(* 
:Description: This function block is used represent basic axis controled by standard PLCopen motion function blocks with collision avoidance feature.
*)
FUNCTION_BLOCK FB_AxisServoCA EXTENDS FB_AxisServo IMPLEMENTS I_UniversalAxisCA
VAR
	(*Commands *)
	bHaltCA				: BOOL;	(*  *)
	bMoveAbsoluteCA		: BOOL;	(*  *)
	bMoveRelativeCA		: BOOL;	(*  *)
	bHaltedCA			: BOOL;
	
	(* Parameters *)
	lrGap				: MC_LREAL;
	eDirectionCa		: Tc3_Mc3Definitions.MC_DIRECTION; (* Axis movement direction for collision avoidance *)
	stMoveAbsCaOptions	: ST_MoveAbsoluteCAOptions;
		
	(* Function blocks *)
	fbMcHaltCA			: MC_HaltCA;			(* Halt with colision avoidance *)
	fbMcMoveAbsoluteCA	: MC_MoveAbsoluteCA;	(* Move absolute with colision avoidance *)
	fbMcMoveRelativeCA	: MC_MoveRelativeCA;	(* Move relative with colision avoidance *)
	
	eAxisStateCA		: E_AxisStateCA;		(*  *)
	tonDelay			: TON;				(* Delay which allows to see any page changes during tests *)

END_VAR
(*
Version history:

+-------------+------------+----------------+----------+------------------------------------------+
|Date         | Version    | created under  | Author   | Remark                                   |
+=============+============+================+==========+==========================================+
|2021-11      | 1.0.0.0    | V3.1.4024.22   | ADBO     | Function block created                   |
+-------------+------------+----------------+----------+------------------------------------------+

*)

IF bFirstCycle THEN
	stMoveAbsCaOptions.GapControlMode := MC_GAP_CONTROL_MODE.mcGapControlModeStandard;
END_IF

SUPER^();

tonDelay();

PROPERTY DirectionCA : Tc3_Mc3Definitions.MC_DIRECTION
GET
DirectionCA := eDirectionCa;
END_GET
SET
eDirectionCa := DirectionCA;
END_SET
END_PROPERTY

PROPERTY Gap : MC_LREAL
GET
Gap := lrGap;
END_GET
SET
lrGap := Gap;
END_SET
END_PROPERTY

PROPERTY HaltedCA : REFERENCE TO BOOL
GET
HaltedCA REF= bHaltedCA;
END_GET
END_PROPERTY

METHOD MR_HaltCA : BOOL
VAR_INPUT
END_VAR
IF eAxisState >= AXIS_IDLE AND eAxisStateCA <> AXIS_CA_HALT_DONE THEN
	bHaltedCA := FALSE;
	
	IF NOT bHaltLog THEN 
		fbMachineLogger.MR_AddLogs(CONCAT(sName,' : halt (CA) requested'));
		bHaltLog := TRUE;
	END_IF
	
	bHaltCA := TRUE;
	MR_HaltCA := FALSE;
	eAxisState := AXIS_EXTENSION;
	eAxisStateCA := AXIS_CA_HALT;
	
ELSIF eAxisState = AXIS_EXTENSION AND eAxisStateCA = AXIS_CA_HALT_DONE THEN
	bInPostion 	:= FALSE;
	bInVelocity := FALSE;
	bMoveActive := FALSE;
	bStopped 	:= FALSE;
	bJogDone 	:= FALSE;
	bHaltedCA	:= TRUE;
	
	bHaltCA		:= FALSE;
	MR_HaltCA 	:= TRUE;
	bHaltLog 	:= FALSE;
	fbMachineLogger.MR_AddLogs(CONCAT(sName,' : halt (CA) done'));
	
END_IF
END_METHOD

METHOD MR_MoveAbsoluteCA : BOOL
VAR_INPUT
	lrAbsolutePosition : LREAL;
END_VAR
VAR
	bFirstCycle		   : BOOL := TRUE;
END_VAR
VAR_INST
	lrAbsolutePositionTemp : LREAL;
END_VAR
IF bFirstCycle THEN
	bFirstCycle := FALSE;
	
	IF THIS^.lrAbsolutePosition = lrAbsolutePosition THEN
		lrAbsolutePositionTemp := lrAbsolutePosition - 0.001;
		
	ELSE
		lrAbsolutePositionTemp := lrAbsolutePosition;
		
	END_IF
END_IF


IF eAxisState = AXIS_IDLE AND THIS^.lrAbsolutePosition <> lrAbsolutePositionTemp THEN
	THIS^.lrAbsolutePosition := lrAbsolutePosition;
	bInPostion 	:= FALSE;
	bInVelocity := FALSE;
	bMoveActive := TRUE;
	bStopped 	:= FALSE;
	bHalted 	:= FALSE;
	bJogDone 	:= FALSE;
	bHaltedCA 	:= FALSE;
	
	bMoveAbsoluteCA := TRUE;
	MR_MoveAbsoluteCA := FALSE;
	eAxisState := AXIS_EXTENSION;
	eAxisStateCA := AXIS_CA_MOVE_ABSOLUTE;
	fbMachineLogger.MR_AddLogs(CONCAT(sName,' : move absoulte (CA) requested'));		
	
ELSIF eAxisState = AXIS_EXTENSION AND eAxisStateCA = AXIS_CA_MOVE_ABSOLUTE_DONE THEN
	bInPostion 		:= TRUE;
	bInVelocity		:= FALSE;
	bMoveActive 	:= FALSE;
	bStopped 		:= FALSE;
	bHalted			:= FALSE;
	bJogDone 		:= FALSE;
	bHaltedCA 		:= TRUE;
	
	bMoveAbsoluteCA := FALSE;
	MR_MoveAbsoluteCA := TRUE;
	fbMachineLogger.MR_AddLogs(CONCAT(sName,' : move absoulte (CA) done'));		
	
END_IF
END_METHOD

METHOD MR_MoveRelativeCA : BOOL
VAR_INPUT
	lrRelativeDistance : LREAL;
END_VAR
IF eAxisState = AXIS_IDLE AND lrRelativeDistance <> 0.0 THEN
	bInPostion 	:= FALSE;
	
	THIS^.lrRelativeDistance := lrRelativeDistance;
	bInVelocity := FALSE;
	bMoveActive := TRUE;
	bStopped 	:= FALSE;
	bHalted 	:= FALSE;
	bJogDone 	:= FALSE;
	bHaltedCA 	:= FALSE;
	
	bMoveRelativeCA := TRUE;
	MR_MoveRelativeCA := FALSE;
	eAxisState := AXIS_EXTENSION;
	eAxisStateCA := AXIS_CA_MOVE_RELATIVE;
	fbMachineLogger.MR_AddLogs(CONCAT(sName,' : move relative (CA) requested'));			
	
ELSIF eAxisState = AXIS_EXTENSION AND eAxisStateCA = AXIS_CA_MOVE_RELATIVE_DONE THEN
	bInVelocity 	:= FALSE;
	bMoveActive 	:= FALSE;
	bStopped 		:= FALSE;
	bHalted 		:= FALSE;
	bJogDone 		:= FALSE;
	bHaltedCA 		:= TRUE;
	
	bMoveRelativeCA := FALSE;
	MR_MoveRelativeCA := TRUE;
	bInPostion 		:= TRUE;
	fbMachineLogger.MR_AddLogs(CONCAT(sName,' : move relative (CA) done'));		
	
END_IF
END_METHOD

METHOD PROTECTED MS_Aborting
VAR_INPUT
END_VAR
(* Reset MC_MoveAbsoluteCA *)
fbMcMoveAbsoluteCA( Axis := stAxisRef, Execute := FALSE);

(* Reset MC_MoveRelativeCA *)
fbMcMoveRelativeCA( Axis := stAxisRef, Execute := FALSE);

(* Reset MC_HaltCA *)
fbMcHaltCA( Axis := stAxisRef, Execute := FALSE);

(* Run parent deinitializing procedure *)
SUPER^.MS_Aborting();
END_METHOD

METHOD MS_AxisCAIdle : BOOL
VAR_INPUT
END_VAR
;
END_METHOD

METHOD MS_Extension : BOOL
VAR_INPUT
END_VAR
CASE eAxisStateCA OF
	E_AxisStateCA.AXIS_CA_IDLE:
		MS_AxisCAIdle();
		
	E_AxisStateCA.AXIS_CA_MOVE_ABSOLUTE:
		MS_MoveAbsoluteCA();
		
	E_AxisStateCA.AXIS_CA_MOVE_ABSOLUTE_DONE:
		MS_MoveAbsoluteCADone();
		
	E_AxisStateCA.AXIS_CA_MOVE_RELATIVE:
		MS_MoveRelativeCA();
		
	E_AxisStateCA.AXIS_CA_MOVE_RELATIVE_DONE:
		MS_MoveRelativeCADone();
		
	E_AxisStateCA.AXIS_CA_HALT:
		MS_HaltCA();
		
	E_AxisStateCA.AXIS_CA_HALT_DONE:
		MS_HaltDoneCA();
	
END_CASE
END_METHOD

METHOD PROTECTED MS_HaltCA
VAR_INPUT
END_VAR
fbMcHaltCA( Axis			:= stAxisRef,
			Execute			:= TRUE,
			Deceleration	:= lrDeceleration,
			Gap				:= lrGap);
	
IF fbMcHaltCA.Error THEN
	bError := TRUE;
	iErrorID := fbMcHaltCA.ErrorId;
	fbMcHaltCA( Axis := stAxisRef, Execute := FALSE);	
	fbAlarmHaltCA.ipArguments.Clear().AddUDInt(iErrorID);	
	fbAlarmHaltCA.Raise(0);

ELSIF fbMcHaltCA.Done THEN
	fbMcMoveAbsoluteCA( Axis := stAxisRef, Execute := FALSE);
	eAxisStateCA := AXIS_CA_HALT_DONE;
	bHalted 	:= TRUE;
	
END_IF
END_METHOD

METHOD PROTECTED MS_HaltDoneCA
VAR_INPUT
END_VAR
(* Reset MC_HaltCA *)
fbMcHaltCA( Axis := stAxisRef, Execute := FALSE);	

IF NOT bHaltCA AND NOT fbMcHaltCA.Busy THEN
	tonDelay(IN := TRUE, PT:= T#200MS);
	
	IF tonDelay.Q THEN
		tonDelay(IN := FALSE);
		eAxisState := AXIS_IDLE;
		eAxisStateCA := AXIS_CA_IDLE;
		
	END_IF
END_IF
END_METHOD

METHOD MS_MoveAbsoluteCA : BOOL
VAR_INPUT
END_VAR
CASE eAxesGroupMethodState OF
	AXES_GROUP_METHOD_EXECUTE:
		fbMcMoveAbsoluteCA(	Axis			:= stAxisRef,
							Execute			:= TRUE,
							Velocity		:= lrVelocity,
							Position		:= lrAbsolutePosition,
							Acceleration	:= lrAcceleration,
							Deceleration	:= lrDeceleration,
							Jerk			:= lrJerk,
							Gap				:= lrGap,
							Direction		:= eDirectionCa,
							Options			:= stMoveAbsCaOptions);

		IF NOT fbMcMoveAbsoluteCA.Busy THEN
			eAxesGroupMethodState := AXES_GROUP_METHOD_DONE; 
			
		END_IF
	
	AXES_GROUP_METHOD_DONE:
		IF fbMcMoveAbsoluteCA.Error THEN
			bError := TRUE;
			iErrorID := fbMcMoveAbsoluteCA.ErrorId;
			fbMcMoveAbsoluteCA( Axis := stAxisRef, Execute := FALSE);
			fbAlarmMoveAbsoluteCA.ipArguments.Clear().AddUDInt(iErrorID);
			fbAlarmMoveAbsoluteCA.Raise(0);
				
		ELSE //fbMcMoveAbsoluteCA.Done THEN
			eAxisStateCA := AXIS_CA_MOVE_ABSOLUTE_DONE;
			
		END_IF
END_CASE
END_METHOD

METHOD MS_MoveAbsoluteCADone : BOOL
VAR_INPUT
END_VAR
(* Reset MC_MoveAbsoluteCA *)
fbMcMoveAbsoluteCA( Axis := stAxisRef, Execute := FALSE);

IF bInPostion THEN
	eAxisState := AXIS_IDLE;
 	eAxesGroupMethodState := AXES_GROUP_METHOD_EXECUTE;
	eAxisStateCA := AXIS_CA_IDLE;
	
END_IF
END_METHOD

METHOD PROTECTED MS_MoveRelativeCA
VAR_INPUT
END_VAR
CASE eAxesGroupMethodState OF
	AXES_GROUP_METHOD_EXECUTE:
		fbMcMoveRelativeCA(	Axis			:= stAxisRef,
							Execute			:= TRUE,
							Distance		:= lrRelativeDistance,
							Velocity		:= lrVelocity,
							Acceleration	:= lrAcceleration,
							Deceleration	:= lrDeceleration,
							Jerk			:= lrJerk,
							Gap 			:= lrGap);

		IF NOT fbMcMoveRelativeCA.Busy THEN
			eAxesGroupMethodState := AXES_GROUP_METHOD_DONE; 
			
		END_IF
							
							
	AXES_GROUP_METHOD_DONE:						
		IF fbMcMoveRelativeCA.Error THEN
			bError := TRUE;
			iErrorID := fbMcMoveRelativeCA.ErrorId;
			fbMcMoveRelativeCA( Axis := stAxisRef, Execute := FALSE);
			fbAlarmMoveRelativeCA.ipArguments.Clear().AddUDInt(iErrorID);
			fbAlarmMoveRelativeCA.Raise(0);
			
		ELSE //fbMcMoveRelativeCA.Done THEN
			eAxisStateCA := AXIS_CA_MOVE_RELATIVE_DONE;
				
		END_IF
END_CASE
END_METHOD

METHOD PROTECTED MS_MoveRelativeCADone
VAR_INPUT
END_VAR
(* Reset MC_MoveRelativeCA *)
fbMcMoveRelativeCA( Axis := stAxisRef, Execute := FALSE);

IF bInPostion THEN
	eAxisState := AXIS_IDLE;
	eAxisStateCA := AXIS_CA_IDLE;
 	eAxesGroupMethodState := AXES_GROUP_METHOD_EXECUTE;

END_IF
END_METHOD

(* 
Copyrights	: Sonion Industrialization - Control Systems Desing Department
Author		: Adrian Bogdzia - based on MEMS universal libraries
Date		: 11/2021
Description : This function block is used represent basic axis
*)
METHOD PROTECTED MS_Reset
VAR_INPUT
END_VAR
(* Reset MC_MoveAbsoluteCA *)
fbMcMoveAbsoluteCA( Axis := stAxisRef, Execute := FALSE);

(* Reset MC_MoveRelativeCA *)
fbMcMoveRelativeCA( Axis := stAxisRef, Execute := FALSE);

(* Reset MC_HaltCA *)
fbMcHaltCA( Axis := stAxisRef, Execute := FALSE);

(* Run parent reset procedure *)
SUPER^.MS_Reset();
END_METHOD

METHOD PROTECTED MS_Stop
VAR_INPUT
END_VAR
(* Reset MC_MoveAbsoluteCA *)
fbMcMoveAbsoluteCA( Axis := stAxisRef, Execute := FALSE);

(* Reset MC_MoveRelativeCA *)
fbMcMoveRelativeCA( Axis := stAxisRef, Execute := FALSE);

(* Run parent stop procedure *)
SUPER^.MS_Stop();
END_METHOD

PROPERTY StateCA : REFERENCE TO E_AxisStateCA
GET
StateCA REF= eAxisStateCA;
END_GET
END_PROPERTY

END_FUNCTION_BLOCK

(* stored: Version 1.1.0.1, ProductVersion 3.1.4024.12
   POU FB_AxisServoCA: Id {9c7dd025-1ca4-413b-8adb-df7153fb7e92}, SpecialFunc None
   Folder Properties: Id {182c7b33-2cc7-49f2-814e-46b99b871fe1}
   Folder Requests: Id {d8238247-8f21-4860-8846-e3ea20f17e20}
   Folder StateMachine: Id {4a5c2a01-6411-4f7e-8f96-78ec3edac617}
   Property DirectionCA: Id {9901e8e7-8dea-40de-bd99-e0c77a372667}
   Get Get: Id {0190fe7f-8401-4dae-ad3c-d21a3c30d810}
   Set Set: Id {0efe00c0-af9b-43fb-acbd-fcac5d4698a9}
   Property Gap: Id {ad665404-c9a6-4f2c-add6-21cbabb4e4c4}
   Get Get: Id {a5713067-08d8-4d9d-8404-3931b1941e41}
   Set Set: Id {758ea178-3b11-4f96-ace7-e0dd2b0aa772}
   Property HaltedCA: Id {143ea7ed-96c5-442f-9629-04b14b1f274c}
   Get Get: Id {f9828fd1-5ce1-44f5-a709-49d3346e84b6}
   Method MR_HaltCA: Id {7e38ff9c-0421-43d1-b647-2364e47bd367}
   Method MR_MoveAbsoluteCA: Id {ee6c5c7f-d50b-4d28-98e2-eea3abdaf044}
   Method MR_MoveRelativeCA: Id {d5bc28a8-c0ff-4391-9dc4-202616c69198}
   Method MS_Aborting: Id {fd5ca5c3-0e71-4cda-b929-a862823a674f}
   Method MS_AxisCAIdle: Id {2eaca4f8-70d9-44fd-a98a-5bbfea9ad285}
   Method MS_Extension: Id {c07209f4-02f9-40da-b1e1-2c0a5a710676}
   Method MS_HaltCA: Id {471b9f5e-06f4-4aca-aa53-292d806a2be3}
   Method MS_HaltDoneCA: Id {a258ad4b-21e9-45d8-b8c1-9fa114108b0c}
   Method MS_MoveAbsoluteCA: Id {4694601e-b888-427c-93e0-b93e725bc1e0}
   Method MS_MoveAbsoluteCADone: Id {5fd94a87-7a7a-43b4-93cf-28771c9e1d96}
   Method MS_MoveRelativeCA: Id {74fe9a71-040a-48fe-ab64-3542140db805}
   Method MS_MoveRelativeCADone: Id {45de7420-0263-4dc3-990b-1c737d0add5f}
   Method MS_Reset: Id {f7516fcf-e88a-46da-b134-63ef8840718f}
   Method MS_Stop: Id {073c3e6a-169c-4154-b6bb-112497bee1aa}
   Property StateCA: Id {9c8a5cf4-b44c-4be0-bd32-f881796a97b3}
   Get Get: Id {37d4f398-0629-4bad-b95f-ed76a0adc1ad} *)
